{attribute 'GeneratedUsingTerminal: EL3773-0000-0016'}
{attribute addProperty BoxType "EL3773-0000-0016"}
{attribute addProperty Id "Cycle_CountAT %I*UINT2"}
{attribute addProperty CRC "2980656546"}
{attribute addProperty Size "2"}
TYPE AI_CycleCount_B1A935A2 :
STRUCT
	{attribute addProperty Name "Cycle_Count"}
	Cycle_Count AT %I* : UINT;
END_STRUCT
END_TYPE

(* stored: Version 1.2.0.0, ProductVersion 3.1.4024.9
   DUT AI_CycleCount_B1A935A2: Id {3c0ec9ba-11dc-4c59-9f90-20f8e178d22b} *)
